// TwinCAT 3 PLC project Bronkhorst
// Title: ZigaLibs.Bronkhorst
// Company: Ziga Javornik
// Author: Ziga Javornik
// ProjectVersion: 0.0.3.1
// Description: Various bronkhorst device impleentations.
// ProgramVersion: 3.1.4026.26
// libraries:
//   Tc2_Standard, * (Beckhoff Automation GmbH)
//   Tc2_System, * (Beckhoff Automation GmbH)
//   Tc3_Module, * (Beckhoff Automation GmbH)
//   TcUnit, * (www.tcunit.org)
//   ZigaLibs.Core, * (Ziga Javornik)
//   ZigaLibs.Logging, * (Ziga Javornik)
// project tree:
//   SOURCE/ FlowUnits.TcPOU (not stored), GasTypes.TcPOU
//   SOURCE/MassFlow or PressureController/DUTs/ E_ControllerMode.TcDUT (not stored), E_ParameterReadingStep.TcDUT (not stored), ST_ControllerCoeList.TcDUT (not stored), ST_ControllerInputs.TcDUT, ST_ControllerOutputs.TcDUT, ST_ControllerStatus.TcDUT (not stored)
//   SOURCE/MassFlow or PressureController/POUs/ FB_FlowController.TcPOU (not stored)
//   / TestsTask.TcTTO (not stored)
//   TESTS/ PRG_TESTS.TcPOU (not stored)
//   TESTS/Test suites/ FB_FlowController_Tests.TcPOU (not stored), FB_FlowUnits_Tests.TcPOU (not stored), FB_GasTypes_Tests.TcPOU (not stored)

// ---- SOURCE/MassFlow or PressureController/DUTs/ST_ControllerInputs.TcDUT
TYPE ST_ControllerInputs :
STRUCT
	MeassuredValue	: INT;
	ValvePosition	: UINT;
	StatusWord		: UINT;
	AmsAddr			: Tc2_System.ST_AmsAddr;
END_STRUCT
END_TYPE

// ---- SOURCE/MassFlow or PressureController/DUTs/ST_ControllerOutputs.TcDUT
TYPE ST_ControllerOutputs :
STRUCT
	ControlByte	: USINT;
	Setpoint	: INT;
END_STRUCT
END_TYPE

// ---- SOURCE/GasTypes.TcPOU
{attribute 'no_explicit_call' := 'Body contains no logic, calling methods only allowed.'}
{attribute 'hide_all_locals'}

// A class containing possible gas types for Bronkhorst devices stored as a string.
PROGRAM GasTypes
VAR
END_VAR

{attribute 'monitoring':='call}
PROPERTY Air : STRING
GET
Air := 'AiR';
END_GET
END_PROPERTY

{attribute 'monitoring':='variable'}
PROPERTY BBr3 : STRING
GET
BBr3 := 'BBr3';
END_GET
END_PROPERTY

{attribute 'monitoring':='variable'}
PROPERTY BCl3 : STRING
GET
BCl3 := 'BCl3';
END_GET
END_PROPERTY

{attribute 'monitoring':='variable'}
PROPERTY C2F6 : STRING
GET
C2F6 := 'C2F6';
END_GET
END_PROPERTY

{attribute 'monitoring':='variable'}
PROPERTY Cl2 : STRING
GET
Cl2 := 'Cl2';
END_GET
END_PROPERTY

{attribute 'monitoring':='variable'}
PROPERTY H2 : STRING
GET
H2 := 'H2';
END_GET
END_PROPERTY

{attribute 'monitoring':='variable'}
PROPERTY He : STRING
GET
He := 'He';
END_GET
END_PROPERTY

{attribute 'monitoring':='variable'}
PROPERTY N2 : STRING
GET
N2 := 'N2';
END_GET
END_PROPERTY

{attribute 'monitoring':='variable'}
PROPERTY O2 : STRING
GET
O2 := 'O2';
END_GET
END_PROPERTY

{attribute 'monitoring':='variable'}
PROPERTY SF6 : STRING
GET
SF6 := 'SF6';
END_GET
END_PROPERTY

{attribute 'monitoring':='variable'}
PROPERTY SiF4 : STRING
GET
SiF4 := 'SiF4';
END_GET
END_PROPERTY

END_PROGRAM
